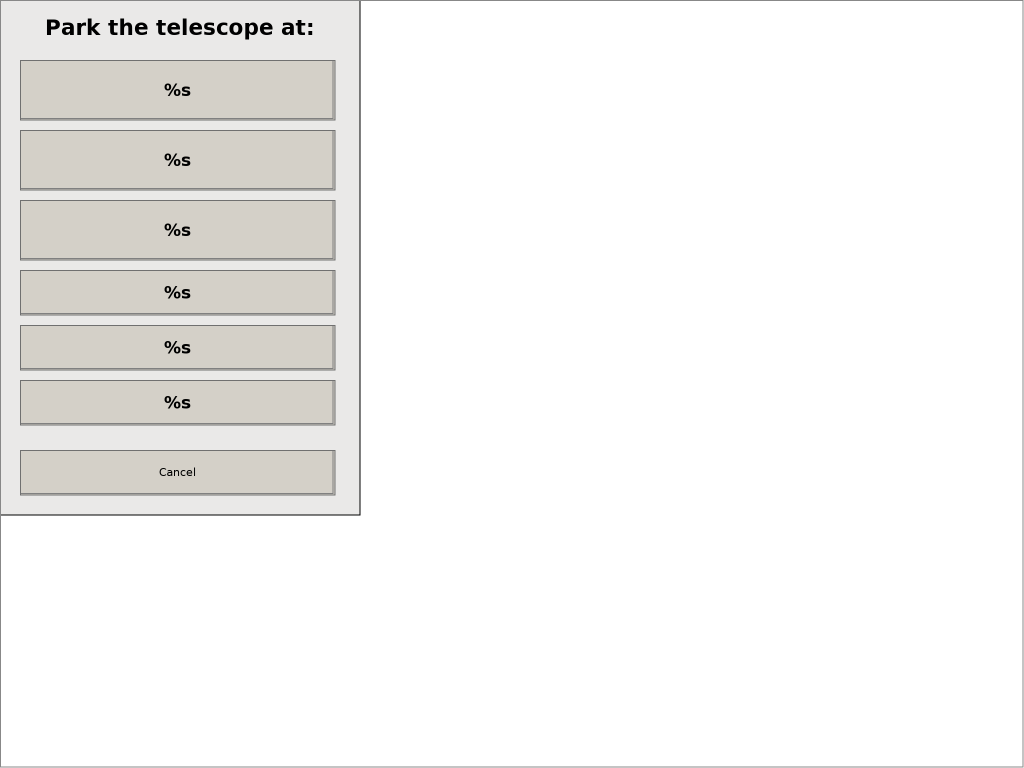
VISUALIZATION VISU_MTCSParkTelescopeDialog  // 1024x768
    Rectangle (0,0 360x515)
    Button (20,60 315x60), "%s", text variable: GLOBAL.mtcs.parts.axes.config.knownPositions.position0.name, invisible if: GLOBAL.gui.axes.manual.positions.invisiblePosition0, input disabled if: GLOBAL.mtcs.parts.axes.processes.moveKnownPosition.statuses.enabledStatus.disabled
        OnMouseClick: execute { GLOBAL.mtcs.parts.axes.processes.moveKnownPosition.request(name := GLOBAL.mtcs.parts.axes.config.knownPositions.position0.name); }
        OnMouseClick: CloseDialog Dialog=VISU_MTCSParkTelescopeDialog, Result=OK, NumpadKeypadSet=True
    Label (0,5 360x45), "Park the telescope at:"
    Button (20,450 315x45), "Cancel"
        OnMouseClick: CloseDialog Dialog=VISU_MTCSParkTelescopeDialog, Result=OK, NumpadKeypadSet=True
    Button (20,130 315x60), "%s", text variable: GLOBAL.mtcs.parts.axes.config.knownPositions.position1.name, invisible if: GLOBAL.gui.axes.manual.positions.invisiblePosition1, input disabled if: GLOBAL.mtcs.parts.axes.processes.moveKnownPosition.statuses.enabledStatus.disabled
        OnMouseClick: execute { GLOBAL.mtcs.parts.axes.processes.moveKnownPosition.request(name := GLOBAL.mtcs.parts.axes.config.knownPositions.position1.name); }
        OnMouseClick: CloseDialog Dialog=VISU_MTCSParkTelescopeDialog, Result=OK, NumpadKeypadSet=True
    Button (20,200 315x60), "%s", text variable: GLOBAL.mtcs.parts.axes.config.knownPositions.position2.name, invisible if: GLOBAL.gui.axes.manual.positions.invisiblePosition2, input disabled if: GLOBAL.mtcs.parts.axes.processes.moveKnownPosition.statuses.enabledStatus.disabled
        OnMouseClick: execute { GLOBAL.mtcs.parts.axes.processes.moveKnownPosition.request(name := GLOBAL.mtcs.parts.axes.config.knownPositions.position2.name); }
        OnMouseClick: CloseDialog Dialog=VISU_MTCSParkTelescopeDialog, Result=OK, NumpadKeypadSet=True
    Button (20,270 315x45), "%s", text variable: GLOBAL.mtcs.parts.axes.config.knownPositions.position3.name, invisible if: GLOBAL.gui.axes.manual.positions.invisiblePosition3, input disabled if: GLOBAL.mtcs.parts.axes.processes.moveKnownPosition.statuses.enabledStatus.disabled
        OnMouseClick: execute { GLOBAL.mtcs.parts.axes.processes.moveKnownPosition.request(name := GLOBAL.mtcs.parts.axes.config.knownPositions.position3.name); }
        OnMouseClick: CloseDialog Dialog=VISU_MTCSParkTelescopeDialog, Result=OK, NumpadKeypadSet=True
    Button (20,325 315x45), "%s", text variable: GLOBAL.mtcs.parts.axes.config.knownPositions.position0.name, invisible if: GLOBAL.gui.axes.manual.positions.invisiblePosition4, input disabled if: GLOBAL.mtcs.parts.axes.processes.moveKnownPosition.statuses.enabledStatus.disabled
        OnMouseClick: execute { GLOBAL.mtcs.parts.axes.processes.moveKnownPosition.request(name := GLOBAL.mtcs.parts.axes.config.knownPositions.position4.name); }
        OnMouseClick: CloseDialog Dialog=VISU_MTCSParkTelescopeDialog, Result=OK, NumpadKeypadSet=True
    Button (20,380 315x45), "%s", text variable: GLOBAL.mtcs.parts.axes.config.knownPositions.position5.name, invisible if: GLOBAL.gui.axes.manual.positions.invisiblePosition5, input disabled if: GLOBAL.mtcs.parts.axes.processes.moveKnownPosition.statuses.enabledStatus.disabled
        OnMouseClick: execute { GLOBAL.mtcs.parts.axes.processes.moveKnownPosition.request(name := GLOBAL.mtcs.parts.axes.config.knownPositions.position5.name); }
        OnMouseClick: CloseDialog Dialog=VISU_MTCSParkTelescopeDialog, Result=OK, NumpadKeypadSet=True
END_VISUALIZATION

(* stored: Version 1.1.0.1, ProductVersion 3.1.4019.2
   Visu VISU_MTCSParkTelescopeDialog: Id {b7ecda67-ef42-4d97-8764-fa12996a2ad2} *)
